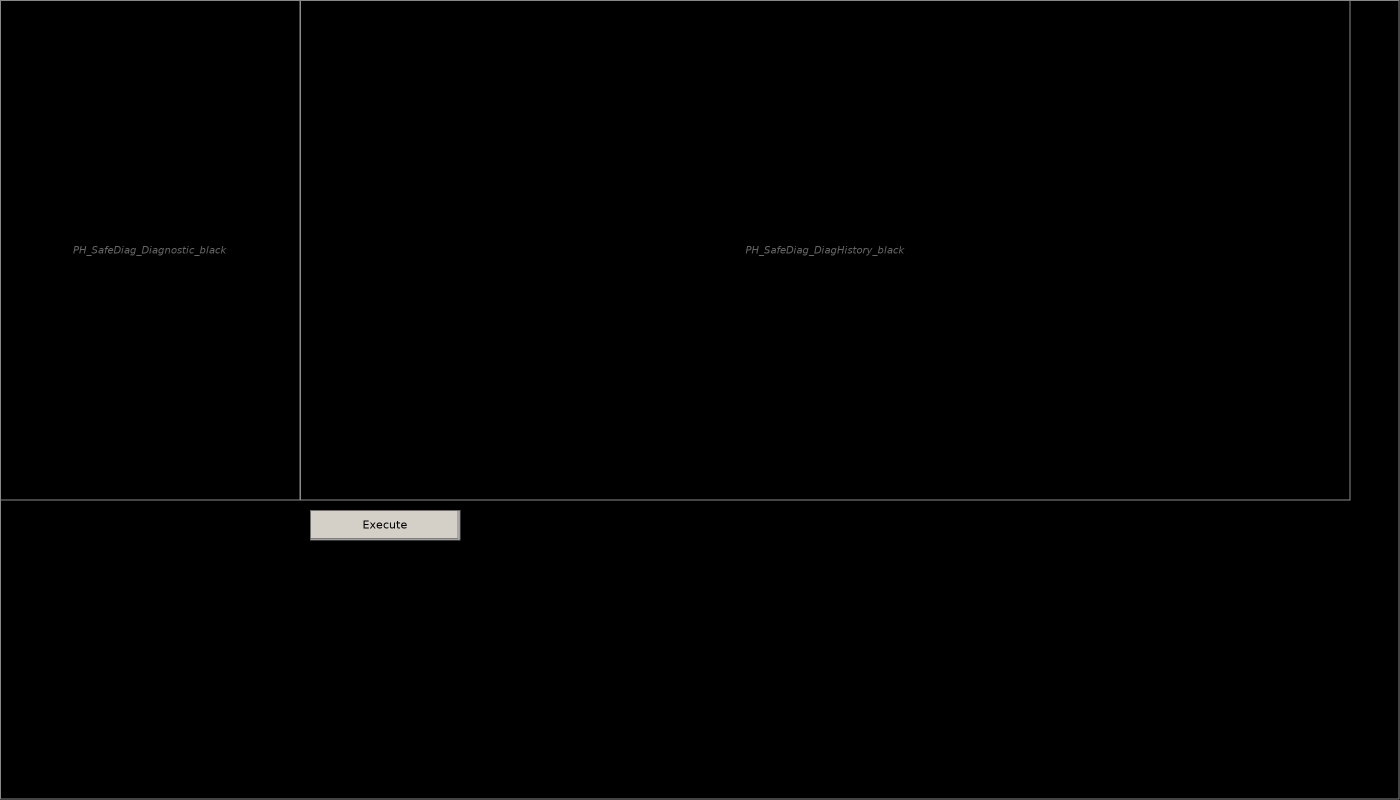
VISUALIZATION V_SafeDiag_Main  // 1400x800
    Button (310,510 150x30), "Execute"
        tap P_Sample.bExecute
    Frame (0,0 300x500)
        shows PH_SafeDiag_Diagnostic_black(stVisu := P_Sample.stSafeDiag.stVisu, stSafeDiag := P_Sample.stSafeDiag)
    Frame (300,0 1050x500)
        shows PH_SafeDiag_DiagHistory_black()
END_VISUALIZATION

(* stored: Version 1.1.0.1, ProductVersion 3.1.4024.12
   Visu V_SafeDiag_Main: Id {1e0c58f3-9237-4f37-b271-33dd1e9e939a} *)
